Fanuc KAREL source: kt00365.KL

-- PROVISIONAL review KL for V770-1; original PC SHA256 eeeafefcbf8a7007953a287e94a29895ec314f9c2fdd9e1888aa3d7566cad458
-- Incomplete behavior may be omitted. Consult companion uncertainty JSON. Do not deploy.
PROGRAM KT00365
%NOLOCKGROUP
VAR
  I1 : INTEGER
  I2 : INTEGER
  OUT : BOOLEAN
BEGIN
  -- UNRESOLVED_PC offsets 5-16; opcodes 2E,23
  -- UNRESOLVED_PC offsets 21-32; opcodes 2E,23
  -- UNRESOLVED_PC offsets 37-48; opcodes 2E,23
  -- UNRESOLVED_PC offsets 53-64; opcodes 2E,23
  -- UNRESOLVED_PC offsets 69-88; opcodes 21,21,5A,23
  -- UNRESOLVED_PC offsets 93-97; opcodes 7F
END KT00365
